{attribute 'enable_dynamic_creation'}
FUNCTION_BLOCK StepManagerBasic IMPLEMENTS IStepManager
VAR
	_currentStep : ENUM;
	_requestNumber : DINT;
END_VAR

METHOD _requestStep : BOOL
VAR_INPUT
	nextStep : ENUM;
END_VAR
_requestNumber := _requestNumber + 1; 
_currentStep := nextStep;
END_METHOD

METHOD _reset : BOOL
_currentStep := SEQUENCE_STEP.NO_STEP;
END_METHOD

METHOD _sequenceComplete : BOOL
_requestNumber := _requestNumber + 1; 
_currentStep := SEQUENCE_STEP.NO_STEP;
END_METHOD

METHOD _sequenceError : BOOL
_requestNumber := _requestNumber + 1; 
_currentStep := SEQUENCE_STEP.NO_STEP;
END_METHOD

PROPERTY currentStep : ENUM
GET
currentStep := _currentStep;
END_GET
END_PROPERTY

{warning 'add property implementation'}
PROPERTY RequestNumber : DINT
GET
RequestNumber := _requestNumber;
END_GET
END_PROPERTY

END_FUNCTION_BLOCK

(* stored: Version 1.1.0.1, ProductVersion 3.1.4024.12
   POU StepManagerBasic: Id {093266f8-f27d-447f-8d0c-4f60d6268941}, SpecialFunc None
   Method _requestStep: Id {631d6933-a3d4-4a04-8d8b-2defab756516}
   Method _reset: Id {fb88c2f8-268f-48f3-8ad4-521cc35aeb3a}
   Method _sequenceComplete: Id {ff6a8092-1516-4df4-b57d-1bb9d4d5c97b}
   Method _sequenceError: Id {a9f4d538-abc7-4246-9047-1ad6d24ed996}
   Property currentStep: Id {29f4d86c-54a1-42a1-8dae-2fa8be71c206}
   Get Get: Id {6ff7d4db-2de2-41e3-931f-d828caaa0f1f}
   Property RequestNumber: Id {56d18034-f9ba-490e-94ec-3c8b604cd6b0}
   Get Get: Id {3d104d88-59e8-4239-891c-6b40240640ee} *)
